{attribute 'GeneratedUsingTerminal: ER7041-0002-0024'}
{attribute addProperty BoxType "ER7041-0002-0024"}
{attribute addProperty Id "EnableBOOL1ResetBOOL1Reduce_torqueBOOL1Digital_output_1BOOL1"}
{attribute addProperty CRC "1607755581"}
{attribute addProperty Size "4"}
TYPE Control_5FD4673D :
STRUCT
	{attribute addProperty Name "Enable"}
	Enable : BOOL;
	{attribute addProperty Name "Reset"}
	Reset : BOOL;
	{attribute addProperty Name "Reduce_torque"}
	Reduce_torque : BOOL;
	{attribute addProperty Name "Digital_output_1"}
	Digital_output_1 : BOOL;
END_STRUCT
END_TYPE

(* stored: Version 1.2.0.0, ProductVersion 3.1.4024.9
   DUT Control_5FD4673D: Id {a36dc17e-2174-485e-ab8f-ffd442e609cf} *)
